TYPE ST_Coord :
STRUCT
	x	:LREAL;
	y	:LREAL;
END_STRUCT
END_TYPE

(* stored: Version 1.1.0.1, ProductVersion 3.1.4024.12
   DUT ST_Coord: Id {52a06245-1716-471f-a02d-dba02328790d} *)
